Staubli VAL3: clkValve4.pgx

program clkValve4()
begin
  call toggleValve(4)
end
